INTERFACE ITF_StartUpSequence

METHOD Call : BOOL
VAR_INPUT
END_VAR
END_METHOD

END_INTERFACE

(* stored: Version 1.1.0.1, ProductVersion 3.1.4024.11
   Itf ITF_StartUpSequence: Id {32d8b04a-f014-491d-afb7-bd5a8ac54278}
   Method Call: Id {50a5adc6-bb16-4844-bc1b-f0820b15f97d} *)
